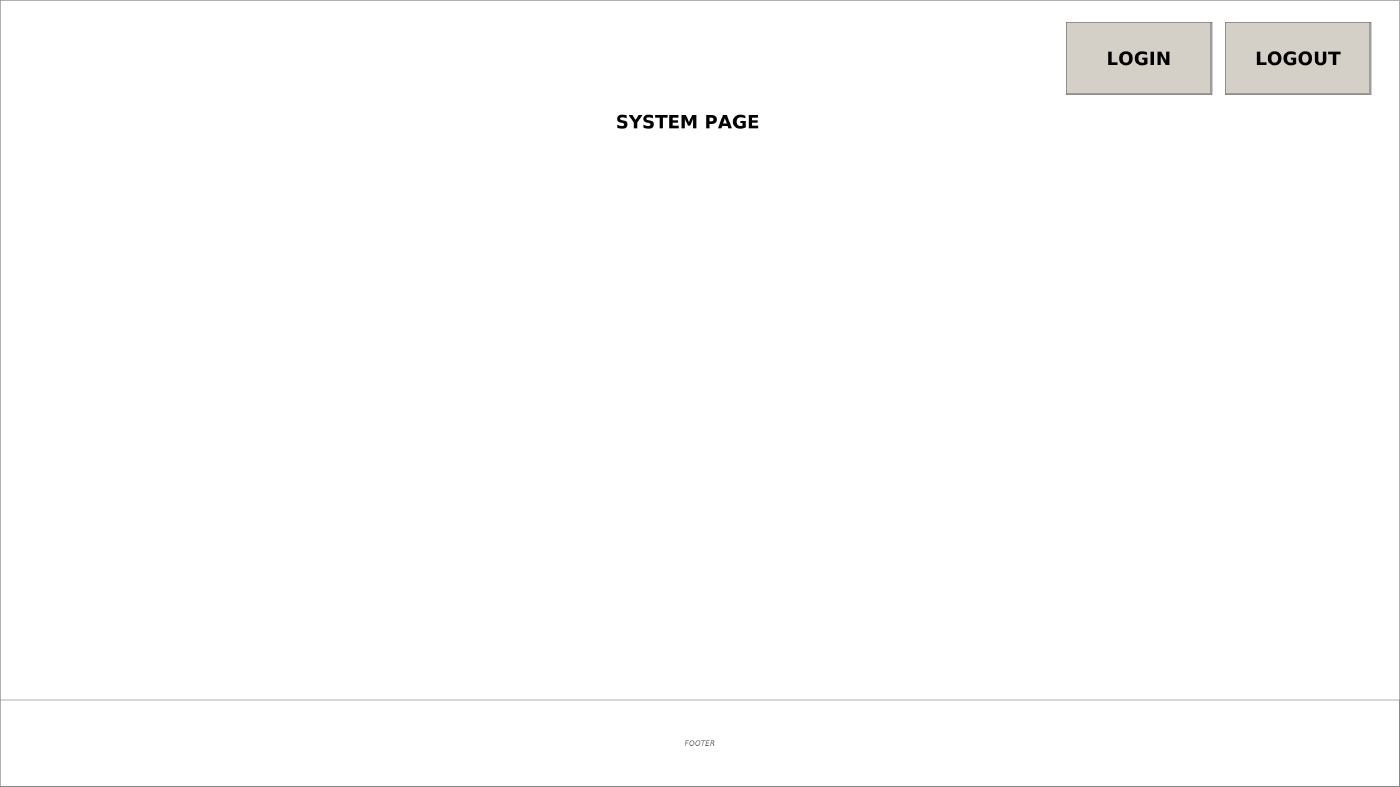
VISUALIZATION PAGE_SYSTEM  // 1920x1080, background image ImagePool.Grey_Gradient
    Button (1462,30 200x100), "LOGIN"
        OnMouseClick: VisuUserMgmt Type=Login
    Button (1680,30 200x100), "LOGOUT"
        OnMouseClick: VisuUserMgmt Type=Logout
    Frame (0,960 1920x120)
        shows FOOTER()
    Label (708,109 470x116), "SYSTEM PAGE"
END_VISUALIZATION

(* stored: Version 1.1.0.1, ProductVersion 3.1.4024.12
   Visu PAGE_SYSTEM: Id {cfc27176-cf48-4ac1-be62-28f63ab99bba} *)
